FUNCTION_BLOCK C_SERIALCOMM_EL6xxx EXTENDS C_SERIALCOMM_PORT
VAR_INPUT
END_VAR
VAR_OUTPUT
END_VAR
VAR
	_hwRxBuffer		AT %I* : EL6inData22B;
	_hwTxBuffer		AT %Q* : EL6outData22B;
END_VAR

METHOD FastBackgroundTask : DINT
{message 'PC type Comm Port implemented'}
C_LINECONTROL(
	Mode:= SERIALLINEMODE_EL6_22B, 
	pComIn:= ADR(_hwRxBuffer), 
	pComOut:= ADR(_hwTxBuffer), 
	SizeComIn:= SIZEOF(_hwRxBuffer), 
	TxBuffer:= _txbuffer, 
	RxBuffer:= _rxbuffer);
END_METHOD

END_FUNCTION_BLOCK

(* stored: Version 1.1.0.1, ProductVersion 3.1.4019.2
   POU C_SERIALCOMM_EL6xxx: Id {d8ebae4b-5429-44ab-95ab-60e002b19f0f}, SpecialFunc None
   Method FastBackgroundTask: Id {e8e24661-1946-404e-81cc-392f7b282ea5} *)
